PROGRAM IOSTATE
VAR
END_VAR


(*EL1859-1 & EL1859-2 STATE*)
IF MOBILEHOIST.IOSTATE1 = FALSE OR MOBILEHOIST.IOSTATE2 = FALSE THEN
	
	MOBILEHOIST.IOERROR		:= TRUE;
	
ELSE
	
	MOBILEHOIST.IOERROR		:= FALSE;
	
END_IF

END_PROGRAM

(* stored: Version 1.1.0.1, ProductVersion 3.1.4024.11
   POU IOSTATE: Id {98fdfa3a-66f1-4679-a388-28e174bc3086}, SpecialFunc None *)
